RoboDK station: LabMotoman.rdk

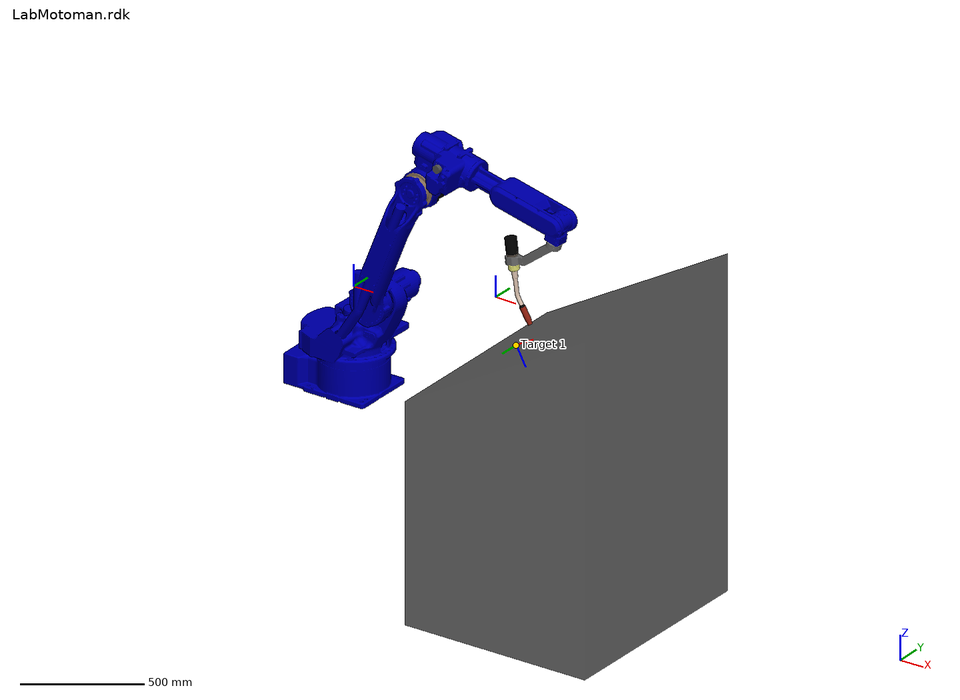
[picture v0: the station drawn from its stored meshes, robots at their saved joint values, targets as dots, program paths as lines]
Station Robodk (2) (saved by RoboDK 5.9.0). Poses are relative to the parent item; angles as X-Y-Z fixed-axis rotations.
  - frame Motoman MH6 Base at (0, 0, 450) mm
    - robot Motoman MH6: 6 axes, payload 6 kg, reach 1422 mm, repeatability 0.08 mm, weight 130 kg
        modified DH rows (alpha deg, a mm, theta deg, d mm): 0, 0, 0, 450; -90, 152, -90, 0; 0, 614, 0, 0; -90, 155, 0, 640; 90, 0, 90, 0; -90, 0, 0, 95
        base shift (0, 0, -450) mm
        joint limits [-170, -90, -175, -180, -45, -360] to [170, 155, 250, 180, 225, 360]; home [0, 0, 0, 0, 0, 0]; saved at [-2.005, 21.787, 9.685, 0.52, -2.888, 1.963]
      - tool Lorch LMR 450 W Welding Gun, TCP at (0, -1.83, 428.17) mm, rotated rx 0 ry 45 rz 0 deg, size 253.4 x 63 x 432.3 mm
    - target Target 1 (Cartesian target) at (823.2, -34.49, -21.13) mm, rotated rx -180 ry -30 rz 0 deg; joints [-2.17, 14.902, -8.252, 0.567, 8.164, 2.016] of Motoman MH6
    - frame Frame_from_Target1 at (823.2, -34.49, -21.13) mm, rotated rx -180 ry -30 rz 0 deg
  - object CAJA2 at (1600, 500, 300) mm, rotated rx 180 ry 0 rz 0 deg, size 886.4 x 1000 x 1511.7 mm, geometry from CAJA2.stp
  - Python program Target_A_Frame (listed below)
  - Python program Espiral (listed below)
  - Python program FigPolar (listed below)
  - Python program HolaFuncional (listed below)
  - frame Frame_from_Target1 at (0, 1000, 0) mm

--- Python program Target_A_Frame ---
from robodk.robolink import *    # API para comunicarte con RoboDK
from robodk.robomath import *    # Mat, Pose_2_TxyzRxyz, etc.

#------------------------------------------------
# 1) Conectar con RoboDK
#------------------------------------------------
RDK = Robolink()

# Tomamos el item "Target1" de la estación, de tipo objetivo (target)
target_item = RDK.Item("Target 1", ITEM_TYPE_TARGET)
if not target_item.Valid():
    raise Exception("No se encontró un Target llamado 'Target1'")

#------------------------------------------------
# 2) Leer la pose y el padre (item padre)
#------------------------------------------------
pose_target = target_item.Pose()  # Matriz 4x4
parent_item = target_item.Parent()  # El padre puede ser el robot base, un frame, etc.

#------------------------------------------------
# 3) Crear un nuevo Frame
#------------------------------------------------
# Le damos un nombre, por ejemplo "Frame_from_Target1"
frame_name = "Frame_from_Target1"
RDK.AddFrame(frame_name)
new_frame = RDK.Item(frame_name, ITEM_TYPE_FRAME)
if not new_frame.Valid():
    raise Exception("No se pudo crear el Frame 'Frame_from_Target1'")

#------------------------------------------------
# 4) Asignar la pose y el mismo padre
#------------------------------------------------
new_frame.setPose(pose_target)     # Copiamos la posición y orientación del target
new_frame.setParent(parent_item)   # Ubicamos el frame bajo el mismo padre que tenía Target1

#------------------------------------------------
# 5) (Opcional) Borrar el Target original
#------------------------------------------------
# target_item.Delete()

print(f"Se ha creado el frame '{frame_name}' con la misma pose que 'Target1'.")

--- Python program Espiral ---
from robodk.robolink import *    # API para comunicarte con RoboDK
from robodk.robomath import *    # Funciones matemáticas
import math

#------------------------------------------------
# 1) Conexión a RoboDK e inicialización
#------------------------------------------------
RDK = Robolink()

# Elegir un robot (si hay varios, aparecerá un popup)
robot = RDK.ItemUserPick("Selecciona un robot", ITEM_TYPE_ROBOT)
if not robot.Valid():
    raise Exception("No se ha seleccionado un robot válido.")

#------------------------------------------------
# 2) Tomar el Frame ya creado en RoboDK
#    (ejemplo: "Frame_from_Target1")
#------------------------------------------------
frame_name = "Frame_from_Target1"
frame_inclinado = RDK.Item(frame_name, ITEM_TYPE_FRAME)
if not frame_inclinado.Valid():
    raise Exception(f'No se encontró el Frame "{frame_name}" en la estación.')

# Configuramos el robot para que use este frame
robot.setPoseFrame(frame_inclinado)
# Usamos la herramienta activa (cambia si necesitas otra)
robot.setPoseTool(robot.PoseTool())

# Ajustes de velocidad y blending
robot.setSpeed(100)   # mm/s
robot.setRounding(5)  # radio de curvatura (blend)

#------------------------------------------------
# 3) Parámetros para la espiral
#------------------------------------------------
num_points = 200       # Número de puntos
turns = 3              # Vueltas de la espiral
spiral_spread = 1.0    # Crecimiento del radio por radian
z_surface = 0          # Z=0 en el Frame, considerado la "superficie"
z_safe = 20            # Altura segura para aproximarse/salir

theta_max = 2 * math.pi * turns

# El centro de la espiral en (x=0, y=0, z=0) relativo al Frame
first_x = 0
first_y = 0
first_z = z_surface

#------------------------------------------------
# 4) Movimiento inicial al centro en altura segura
#------------------------------------------------
robot.MoveJ(transl(first_x, first_y, first_z + z_safe))
robot.MoveL(transl(first_x, first_y, first_z))

#------------------------------------------------
# 5) Recorrer la espiral
#------------------------------------------------
for i in range(1, num_points + 1):
    t = i / num_points
    theta = t * theta_max
    r = spiral_spread * theta

    x = r * math.cos(theta)
    y = r * math.sin(theta)
    z = z_surface

    # Movimiento lineal hacia el siguiente punto
    robot.MoveL(transl(x, y, z))

# Al terminar, subimos para alejarnos de la superficie
robot.MoveL(transl(x, y, z + z_safe))

print(f"¡Espiral completada usando el frame '{frame_name}'!")

--- Python program FigPolar ---
from robodk.robolink import *    # API para comunicarte con RoboDK
from robodk.robomath import *    # funciones matemáticas
import math
import numpy as np


# conexión con RoboDK
RDK = Robolink()

# elegir un robot
robot = RDK.ItemUserPick("Selecciona un robot", ITEM_TYPE_ROBOT)
if not robot.Valid():
    raise Exception("No se ha seleccionado un robot válido.")

# cargar frame (ya existente)
frame_name = "Frame_from_Target1"
frame = RDK.Item(frame_name, ITEM_TYPE_FRAME)
if not frame.Valid():
    raise Exception(f'No se encontró el Frame "{frame_name}" en la estación.')

# asignar frame al robot
robot.setPoseFrame(frame)
# seleccionar herramienta activa
robot.setPoseTool(robot.PoseTool())

# ajustes de velocidad
robot.setSpeed(100)   # mm/s
robot.setRounding(5)  # blending

# parámetros de la figura (curva cardioide)
num_points = 720       # número de puntos
A = 120                # escala
z_surface = 0          # z = 0 en el plano del frame
z_safe = -50           # altura segura


# punto de inicio de la figura en coordenadas polares
r_0 = A*(1 - math.cos(0)*sin(0))

# punto de inicio de la figura en coordenadas cartesianas
x_0 = r_0*math.cos(0)
y_0 = r_0*math.sin(0)

# instrucción para mover el robot al punto de inicio de la figura
robot.MoveJ(transl(x_0, y_0, z_surface + z_safe))

# bajar a la superficie de trabajo (z = 0)
robot.MoveL(transl(x_0, y_0, z_surface))

# dibujar la curva polar

# la curva irá de 0 a 2pi
full_turn = 2*math.pi

for i in range(num_points+1):
    # fracción entre 0 y 1
    t = i / num_points
    # ángulo actual
    theta = full_turn * t

    # calcular r
    r = A*(1 - math.cos(theta)*sin(3*theta))

    # conversión de coordenadas polares a cartesianas
    x = r * math.cos(theta)
    y = r * math.sin(theta)

    # mover linealmente (MoveL) en el plano del frame
    robot.MoveL(transl(x, y, z_surface))

# al terminar, subir de nuevo a la zona segura
robot.MoveL(transl(x_0, y_0, z_surface + z_safe))

print(f"Figura completada.")

--- Python program HolaFuncional ---
from robodk.robolink import *    # API para comunicarse con RoboDK
from robodk.robomath import *    # Operaciones matemáticas
import math

#------------------------------------------------
# 1) Conexión a RoboDK e inicialización
#------------------------------------------------
RDK = Robolink()

# Seleccionar un robot (popup si hay más de uno)
robot = RDK.ItemUserPick("Selecciona un robot", ITEM_TYPE_ROBOT)
if not robot.Valid():
    raise Exception("No se ha seleccionado un robot válido.")

# Conectar al robot físico
if not robot.Connect():
    raise Exception("No se pudo conectar al robot. Verifica que esté en modo remoto y que la configuración sea correcta.")

# Confirmar conexión
if not robot.ConnectedState():
    raise Exception("El robot no está conectado correctamente. Revisa la conexión.")

print("Robot conectado correctamente.")

#------------------------------------------------
# 2) Tomar el Frame inclinado
frame_name = "Frame_from_Target1"
frame_inclinado = RDK.Item(frame_name, ITEM_TYPE_FRAME)
if not frame_inclinado.Valid():
    raise Exception(f"No se encontró el Frame '{frame_name}' o no es de tipo FRAME.")

# Asignamos este frame para los próximos movimientos
robot.setPoseFrame(frame_inclinado)
robot.setPoseTool(robot.PoseTool())

# Ajustes de velocidad y blend
robot.setSpeed(100)      # mm/s
robot.setRounding(5)     # Radio de blend (suavizado)

#------------------------------------------------
# 3) Definición de letras
letter_H = [
    [(0, 0), (0, 30)],     # Línea vertical izquierda
    [(0, 15), (10, 15)],   # Línea horizontal central
    [(10, 0), (10, 30)]    # Línea vertical derecha
]

letter_O = [
    [(0, 0), (0, 30), (10, 30), (10, 0), (0, 0)]  # Contorno rectangular cerrado
]

letter_L = [
    [(0, 30), (0, 0)],     # Línea vertical
    [(0, 0), (10, 0)]      # Línea horizontal inferior
]

letter_A = [
    [(0, 0), (5, 30), (10, 0)],  # Triángulo para la letra A
    [(2, 15), (8, 15)]           # Línea horizontal central
]

letters = {
    'H': letter_H,
    'O': letter_O,
    'L': letter_L,
    'A': letter_A
}

#------------------------------------------------
# 4) Parámetros de escritura
word_to_write = "HOLA"
scale = 1.0
spacing = 15
z_draw = 0
pen_up_dist = 15
start_x = 0
start_y = 0

#------------------------------------------------
# 5) Función para dibujar una letra
def draw_letter(letter, offset_x, offset_y):
    polylines = letters.get(letter, [])
    last_x, last_y = offset_x, offset_y

    for pline in polylines:
        x0 = offset_x + scale*pline[0][0]
        y0 = offset_y + scale*pline[0][1]

        pose_move = eye(4)
        pose_move.setPos([x0, y0, z_draw])
        robot.MoveL(pose_move)

        for pt in pline[1:]:
            x = offset_x + scale*pt[0]
            y = offset_y + scale*pt[1]
            pose_line = eye(4)
            pose_line.setPos([x, y, z_draw])
            robot.MoveL(pose_line)
            last_x, last_y = x, y

    return last_x, last_y

#------------------------------------------------
# 6) Dibujar la palabra
current_x = start_x
current_y = start_y

robot.MoveJ(transl(current_x, current_y, z_draw + pen_up_dist))
robot.MoveL(transl(current_x, current_y, z_draw))

for i, letter in enumerate(word_to_write):
    end_x, end_y = draw_letter(letter, current_x, current_y)

    if i < len(word_to_write)-1:
        next_x = current_x + (10*scale + spacing)
        next_y = current_y

        pose_up = robot.Pose()
        pos_up = pose_up.Pos()
        pos_up[2] += pen_up_dist
        pose_up.setPos(pos_up)
        robot.MoveL(pose_up)

        diagonal_pose = eye(4)
        diagonal_pose.setPos([next_x, next_y, z_draw])
        robot.MoveL(diagonal_pose)

        current_x = next_x
        current_y = next_y

robot.MoveL(transl(current_x, current_y, z_draw + pen_up_dist))
print("¡Escritura terminada en el frame inclinado!")
